RoboDK station: 03 - Palletizing.rdk

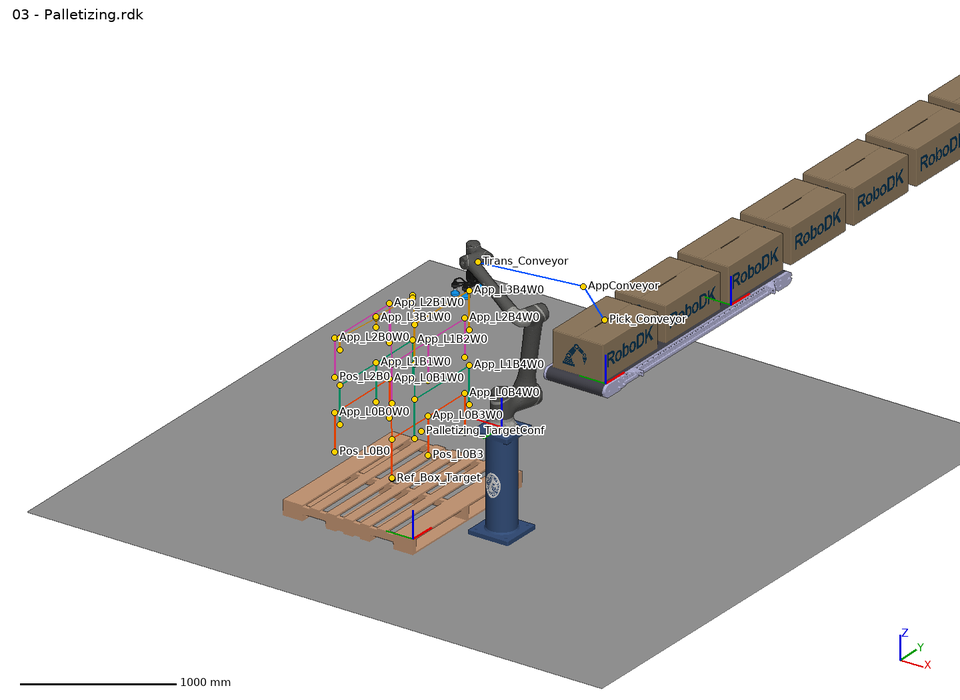
[picture v0: the station drawn from its stored meshes, robots at their saved joint values, targets as dots, program paths as lines]
Station 03 - Palletizing (saved by RoboDK 5.2.4). Poses are relative to the parent item; angles as X-Y-Z fixed-axis rotations.
Station parameters (name, value as stored): Conv_Run, 0, IO_5, 1
  - frame Omron TM12X Base at (0, 0, 0) mm, rotated rx 0 ry 0 rz 180 deg
    - object Pedestal H12in at (0, 0, -305) mm, rotated rx 0 ry 0 rz -90 deg, size 320 x 320 x 304.8 mm, geometry from Pedestal-H12in (2).sld
    - object Pedestal H24in at (0, 0, 0) mm, rotated rx 0 ry 0 rz -180 deg, size 312.1 x 312.1 x 743.1 mm, geometry from Pedestal-H24in.sld
    - object Box 24X16 at (0, 0, 0) mm, size 398.1 x 610.2 x 267.5 mm, geometry from Box 24x16 closed.step
    - robot Omron TM12X: 6 axes, payload 12 kg, reach 1300 mm, repeatability 0.1 mm, weight 33.3 kg
        modified DH rows (alpha deg, a mm, theta deg, d mm): 0, 0, 0, 165.2; 90, 0, 90, 0; 0, 636.1, 0, 0; 0, 557.9, -90, 156.3; -90, 0, 0, 106; 90, 0, 180, 113.15
        joint limits [-125, -90, -60, -145, 0, -200] to [90, 130, 166, 90, 180, 125]; home [0, 0, 90, 0, 90, 0]; saved at [-17.678, -9.72, 76.178, 23.542, 90, -17.678]
      - tool RobotiQ EPick Four, TCP at (0, 30, 180) mm, size 239 x 147 x 184.9 mm
    - frame Conveyor Belt Base at (-430, -550, 210) mm, rotated rx 0 ry 0 rz -90 deg
      - robot Conveyor Belt: 1 axes
          modified DH rows (alpha deg, a mm, theta deg, d mm): 0, 0, 0, 0 linear
          base shift (0, 0, 0) mm, rotated rx 0 ry 90 rz 0 deg
          joint limits [-500000] to [500000]; home [0]; saved at [0]
        - frame Conveyor Box at (0, 0, 0) mm
          - object Box_24X16 at (700, 420, 0) mm, rotated rx 0 ry 0 rz -90 deg, size 398.1 x 610.2 x 267.5 mm, geometry from Box 24x16 closed.step
          - object Box_24X16 at (1400, 420, 0) mm, rotated rx 0 ry 0 rz -90 deg, size 398.1 x 610.2 x 267.5 mm, geometry from Box 24x16 closed.step
          - object Box_24X16 at (5600, 420, 0) mm, rotated rx 0 ry 0 rz -90 deg, size 398.1 x 610.2 x 267.5 mm, geometry from Box 24x16 closed.step
          - object Box_24X16 at (6300, 420, 0) mm, rotated rx 0 ry 0 rz -90 deg, size 398.1 x 610.2 x 267.5 mm, geometry from Box 24x16 closed.step
          - object Box_24X16 at (7700, 420, 0) mm, rotated rx 0 ry 0 rz -90 deg, size 398.1 x 610.2 x 267.5 mm, geometry from Box 24x16 closed.step
          - object Box_24X16 at (7000, 420, 0) mm, rotated rx 0 ry 0 rz -90 deg, size 398.1 x 610.2 x 267.5 mm, geometry from Box 24x16 closed.step
          - object Box_24X16 at (8400, 420, 0) mm, rotated rx 0 ry 0 rz -90 deg, size 398.1 x 610.2 x 267.5 mm, geometry from Box 24x16 closed.step
          - object Box_24X16 at (9100, 420, 0) mm, rotated rx 0 ry 0 rz -90 deg, size 398.1 x 610.2 x 267.5 mm, geometry from Box 24x16 closed.step
          - object Box_24X16 at (10500, 420, 0) mm, rotated rx 0 ry 0 rz -90 deg, size 398.1 x 610.2 x 267.5 mm, geometry from Box 24x16 closed.step
          - object Box_24X16 at (9800, 420, 0) mm, rotated rx 0 ry 0 rz -90 deg, size 398.1 x 610.2 x 267.5 mm, geometry from Box 24x16 closed.step
          - object Box_24X16 at (11200, 420, 0) mm, rotated rx 0 ry 0 rz -90 deg, size 398.1 x 610.2 x 267.5 mm, geometry from Box 24x16 closed.step
          - object Box_24X16 at (11900, 420, 0) mm, rotated rx 0 ry 0 rz -90 deg, size 398.1 x 610.2 x 267.5 mm, geometry from Box 24x16 closed.step
          - object Box_24X16 at (13300, 420, 0) mm, rotated rx 0 ry 0 rz -90 deg, size 398.1 x 610.2 x 267.5 mm, geometry from Box 24x16 closed.step
          - object Box_24X16 at (12600, 420, 0) mm, rotated rx 0 ry 0 rz -90 deg, size 398.1 x 610.2 x 267.5 mm, geometry from Box 24x16 closed.step
          - object Box_24X16 at (0, 420, 0) mm, rotated rx 0 ry 0 rz -90 deg, size 398.1 x 610.2 x 267.5 mm, geometry from Box 24x16 closed.step
          - object Box_24X16 at (2800, 420, 0) mm, rotated rx 0 ry 0 rz -90 deg, size 398.1 x 610.2 x 267.5 mm, geometry from Box 24x16 closed.step
          - object Box_24X16 at (2100, 420, 0) mm, rotated rx 0 ry 0 rz -90 deg, size 398.1 x 610.2 x 267.5 mm, geometry from Box 24x16 closed.step
          - object Box_24X16 at (3500, 420, 0) mm, rotated rx 0 ry 0 rz -90 deg, size 398.1 x 610.2 x 267.5 mm, geometry from Box 24x16 closed.step
          - object Box_24X16 at (4900, 420, 0) mm, rotated rx 0 ry 0 rz -90 deg, size 398.1 x 610.2 x 267.5 mm, geometry from Box 24x16 closed.step
          - object Box_24X16 at (4200, 420, 0) mm, rotated rx 0 ry 0 rz -90 deg, size 398.1 x 610.2 x 267.5 mm, geometry from Box 24x16 closed.step
      - target AppConveyor (Cartesian target) at (69.16, 222.69, 602.66) mm, rotated rx 180 ry 0 rz 179.98 deg; joints [-97.337, 6.658, 49.734, 33.608, 90, -97.317, 0] of Omron TM12X
      - target Pick_Conveyor (Cartesian target) at (304.16, 222.6, 268.74) mm, rotated rx 180 ry 0 rz 179.98 deg; joints [-95.378, 19.16, 70.241, 0.599, 90, -95.357, 0] of Omron TM12X
      - target Trans_Conveyor (Cartesian target) at (-198.64, 863.17, 703.7) mm, rotated rx 180 ry 0 rz -107.24 deg; joints [-25.922, 5.576, 37.342, 47.082, 90, -98.682] of Omron TM12X
      - frame New_Box 24X16 at (1400, 0, 0) mm
        - object BoxRef_24X16 at (0, 420, 0) mm, rotated rx 0 ry 0 rz -90 deg, size 398.1 x 610.2 x 267.5 mm, geometry from Box 24x16 closed.step
    - frame Pallet at (268.35, 609.6, -630.58) mm, rotated rx 0 ry 0 rz -90 deg
      - object Pallet 40inx48in at (0, 0, 0) mm, size 1219.2 x 1016 x 114.3 mm, geometry from AR3.step
      - target Ref_Box_Target (Cartesian target) at (198.15, 304.17, 268.74) mm, rotated rx -180 ry 0 rz -90 deg; joints [46.804, 34.313, 124.082, -68.396, 90, -43.196] of Omron TM12X
      - target Palletizing_TargetConfig (Cartesian target) at (676.2, 408.21, 385.47) mm, rotated rx -179.16 ry 1.93 rz -48.82 deg; joints [5.592, 37.489, 126.42, -75.963, 90.438, -125.563] of Omron TM12X
      - folder Palletizing_Data: PalletData
        - folder Palletizing_Data_L0: PalletData
          - target App_L0B0W0 (Cartesian target) at (303.25, 822.47, 550) mm, rotated rx -180 ry 0 rz -180 deg; joints [24.246, 55.576, 68.456, -34.032, 90, 24.246] of Omron TM12X
          - target Ret_L0B0W0 (Cartesian target) at (303.25, 822.47, 550) mm, rotated rx -180 ry 0 rz -180 deg; joints [24.246, 55.576, 68.456, -34.032, 90, 24.246] of Omron TM12X
          - target Pos_L0B0 (Cartesian target) at (303.25, 822.47, 270) mm, rotated rx -180 ry 0 rz -180 deg; joints [24.246, 73.661, 63.877, -47.538, 90, 24.246] of Omron TM12X
          - target App_L0B1W0 (Cartesian target) at (913.41, 822.47, 550) mm, rotated rx -180 ry 0 rz -180 deg; joints [-7.838, 55.519, 68.577, -34.096, 90, -7.838] of Omron TM12X
          - target Ret_L0B1W0 (Cartesian target) at (913.41, 822.47, 550) mm, rotated rx -180 ry 0 rz -180 deg; joints [-7.838, 55.519, 68.577, -34.096, 90, -7.838] of Omron TM12X
          - target Pos_L0B1 (Cartesian target) at (913.41, 822.47, 270) mm, rotated rx -180 ry 0 rz -180 deg; joints [-7.838, 73.613, 64.003, -47.616, 90, -7.838] of Omron TM12X
          - target App_L0B2W0 (Cartesian target) at (197.9, 303.25, 550) mm, rotated rx -180 ry 0 rz -90 deg; joints [46.878, 30.236, 123.942, -64.178, 90, -43.122] of Omron TM12X
          - target Ret_L0B2W0 (Cartesian target) at (197.9, 303.25, 550) mm, rotated rx -180 ry 0 rz -90 deg; joints [46.878, 30.236, 123.942, -64.178, 90, -43.122] of Omron TM12X
          - target Pos_L0B2 (Cartesian target) at (197.9, 303.25, 270) mm, rotated rx -180 ry 0 rz -90 deg; joints [46.878, 59.272, 119.029, -88.302, 90, -43.122] of Omron TM12X
          - target App_L0B3W0 (Cartesian target) at (604.3, 303.25, 550) mm, rotated rx -180 ry 0 rz -90 deg; joints [13.38, 24.947, 136.655, -71.602, 90, -76.62] of Omron TM12X
          - target Ret_L0B3W0 (Cartesian target) at (604.3, 303.25, 550) mm, rotated rx -180 ry 0 rz -90 deg; joints [13.38, 24.947, 136.655, -71.602, 90, -76.62] of Omron TM12X
          - target Pos_L0B3 (Cartesian target) at (604.3, 303.25, 270) mm, rotated rx -180 ry 0 rz -90 deg; joints [13.38, 60.356, 130.855, -101.211, 90, -76.62] of Omron TM12X
          - target App_L0B4W0 (Cartesian target) at (1015.06, 303.25, 550) mm, rotated rx -180 ry 0 rz -90 deg; joints [-24.738, 31.775, 120.399, -62.175, 90, -114.738] of Omron TM12X
          - target Ret_L0B4W0 (Cartesian target) at (1015.06, 303.25, 550) mm, rotated rx -180 ry 0 rz -90 deg; joints [-24.738, 31.775, 120.399, -62.175, 90, -114.738] of Omron TM12X
          - target Pos_L0B4 (Cartesian target) at (1015.06, 303.25, 270) mm, rotated rx -180 ry 0 rz -90 deg; joints [-24.738, 59.459, 115.654, -85.113, 90, -114.738] of Omron TM12X
        - folder Palletizing_Data_L1: PalletData
          - target App_L1B0W0 (Cartesian target) at (197.9, 709.65, 817.48) mm, rotated rx -180 ry 0 rz -90 deg; joints [29.882, 39.329, 69.189, -18.518, 90, -60.118] of Omron TM12X
          - target Ret_L1B0W0 (Cartesian target) at (197.9, 709.65, 817.48) mm, rotated rx -180 ry 0 rz -90 deg; joints [29.882, 39.329, 69.189, -18.518, 90, -60.118] of Omron TM12X
          - target Pos_L1B0 (Cartesian target) at (197.9, 709.65, 537.48) mm, rotated rx -180 ry 0 rz -90 deg; joints [29.882, 52.141, 77.448, -39.589, 90, -60.118] of Omron TM12X
          - target App_L1B1W0 (Cartesian target) at (604.3, 709.65, 817.48) mm, rotated rx -180 ry 0 rz -90 deg; joints [7.747, 33.003, 80.067, -23.07, 90, -82.253] of Omron TM12X
          - target Ret_L1B1W0 (Cartesian target) at (604.3, 709.65, 817.48) mm, rotated rx -180 ry 0 rz -90 deg; joints [7.747, 33.003, 80.067, -23.07, 90, -82.253] of Omron TM12X
          - target Pos_L1B1 (Cartesian target) at (604.3, 709.65, 537.48) mm, rotated rx -180 ry 0 rz -90 deg; joints [7.747, 47.289, 88.021, -45.31, 90, -82.253] of Omron TM12X
          - target App_L1B2W0 (Cartesian target) at (1015.06, 709.65, 817.48) mm, rotated rx -180 ry 0 rz -90 deg; joints [-15.606, 41.274, 65.737, -17.012, 90, -105.606] of Omron TM12X
          - target Ret_L1B2W0 (Cartesian target) at (1015.06, 709.65, 817.48) mm, rotated rx -180 ry 0 rz -90 deg; joints [-15.606, 41.274, 65.737, -17.012, 90, -105.606] of Omron TM12X
          - target Pos_L1B2 (Cartesian target) at (1015.06, 709.65, 537.48) mm, rotated rx -180 ry 0 rz -90 deg; joints [-15.606, 53.66, 74.159, -37.819, 90, -105.606] of Omron TM12X
          - target App_L1B3W0 (Cartesian target) at (303.25, 200.17, 817.48) mm, rotated rx -180 ry 0 rz -180 deg; joints [51.927, -4.692, 129.582, -34.89, 90, 51.927] of Omron TM12X
          - target Ret_L1B3W0 (Cartesian target) at (303.25, 200.17, 817.48) mm, rotated rx -180 ry 0 rz -180 deg; joints [51.927, -4.692, 129.582, -34.89, 90, 51.927] of Omron TM12X
          - target Pos_L1B3 (Cartesian target) at (303.25, 200.17, 537.48) mm, rotated rx -180 ry 0 rz -180 deg; joints [51.927, 25.107, 140.818, -75.925, 90, 51.927] of Omron TM12X
          - target App_L1B4W0 (Cartesian target) at (913.41, 200.17, 817.48) mm, rotated rx -180 ry 0 rz -180 deg; joints [-17.678, -4.838, 129.711, -34.873, 90, -17.678] of Omron TM12X
          - target Ret_L1B4W0 (Cartesian target) at (913.41, 200.17, 817.48) mm, rotated rx -180 ry 0 rz -180 deg; joints [-17.678, -4.838, 129.711, -34.873, 90, -17.678] of Omron TM12X
          - target Pos_L1B4 (Cartesian target) at (913.41, 200.17, 537.48) mm, rotated rx -180 ry 0 rz -180 deg; joints [-17.678, 25.055, 140.975, -76.03, 90, -17.678] of Omron TM12X
        - folder Palletizing_Data_L2: PalletData
          - target App_L2B0W0 (Cartesian target) at (303.25, 822.47, 1084.96) mm, rotated rx -180 ry 0 rz -180 deg; joints [24.246, 44.227, 32.666, 13.106, 90, 24.246] of Omron TM12X
          - target Ret_L2B0W0 (Cartesian target) at (303.25, 822.47, 1084.96) mm, rotated rx -180 ry 0 rz -180 deg; joints [24.246, 44.227, 32.666, 13.106, 90, 24.246] of Omron TM12X
          - target Pos_L2B0 (Cartesian target) at (303.25, 822.47, 804.96) mm, rotated rx -180 ry 0 rz -180 deg; joints [24.246, 44.92, 60.473, -15.393, 90, 24.246] of Omron TM12X
          - target App_L2B1W0 (Cartesian target) at (913.41, 822.47, 1084.96) mm, rotated rx -180 ry 0 rz -180 deg; joints [-7.838, 44.112, 32.875, 13.013, 90, -7.838] of Omron TM12X
          - target Ret_L2B1W0 (Cartesian target) at (913.41, 822.47, 1084.96) mm, rotated rx -180 ry 0 rz -180 deg; joints [-7.838, 44.112, 32.875, 13.013, 90, -7.838] of Omron TM12X
          - target Pos_L2B1 (Cartesian target) at (913.41, 822.47, 804.96) mm, rotated rx -180 ry 0 rz -180 deg; joints [-7.838, 44.849, 60.603, -15.452, 90, -7.838] of Omron TM12X
          - target App_L2B2W0 (Cartesian target) at (197.9, 303.25, 1084.96) mm, rotated rx -180 ry 0 rz -90 deg; joints [46.878, 0.723, 94.803, -5.526, 90, -43.122] of Omron TM12X
          - target Ret_L2B2W0 (Cartesian target) at (197.9, 303.25, 1084.96) mm, rotated rx -180 ry 0 rz -90 deg; joints [46.878, 0.723, 94.803, -5.526, 90, -43.122] of Omron TM12X
          - target Pos_L2B2 (Cartesian target) at (197.9, 303.25, 804.96) mm, rotated rx -180 ry 0 rz -90 deg; joints [46.878, 9.9, 115.641, -35.541, 90, -43.122] of Omron TM12X
          - target App_L2B3W0 (Cartesian target) at (604.3, 303.25, 1084.96) mm, rotated rx -180 ry 0 rz -90 deg; joints [13.38, -10.122, 104.633, -4.51, 90, -76.62] of Omron TM12X
          - target Ret_L2B3W0 (Cartesian target) at (604.3, 303.25, 1084.96) mm, rotated rx -180 ry 0 rz -90 deg; joints [13.38, -10.122, 104.633, -4.51, 90, -76.62] of Omron TM12X
          - target Pos_L2B3 (Cartesian target) at (604.3, 303.25, 804.96) mm, rotated rx -180 ry 0 rz -90 deg; joints [13.38, -0.241, 126.986, -36.745, 90, -76.62] of Omron TM12X
          - target App_L2B4W0 (Cartesian target) at (1015.06, 303.25, 1084.96) mm, rotated rx -180 ry 0 rz -90 deg; joints [-24.738, 3.601, 91.8, -5.401, 90, -114.738] of Omron TM12X
          - target Ret_L2B4W0 (Cartesian target) at (1015.06, 303.25, 1084.96) mm, rotated rx -180 ry 0 rz -90 deg; joints [-24.738, 3.601, 91.8, -5.401, 90, -114.738] of Omron TM12X
          - target Pos_L2B4 (Cartesian target) at (1015.06, 303.25, 804.96) mm, rotated rx -180 ry 0 rz -90 deg; joints [-24.738, 12.483, 112.359, -34.842, 90, -114.738] of Omron TM12X
        - folder Palletizing_Data_L3: PalletData
          - target App_L3B0W0 (Cartesian target) at (197.9, 709.65, 1150.44) mm, rotated rx -180 ry 0 rz -90 deg; joints [29.882, 38.325, 36.209, 15.467, 90, -60.118] of Omron TM12X
          - target Ret_L3B0W0 (Cartesian target) at (197.9, 709.65, 1158.34) mm, rotated rx -180 ry 0 rz -90 deg; joints [29.882, 38.663, 34.775, 16.561, 90, -60.118] of Omron TM12X
          - target Pos_L3B0 (Cartesian target) at (197.9, 709.65, 1072.44) mm, rotated rx -180 ry 0 rz -90 deg; joints [29.882, 36.374, 47.696, 5.93, 90, -60.118] of Omron TM12X
          - target App_L3B1W0 (Cartesian target) at (604.3, 709.65, 1137.62) mm, rotated rx -180 ry 0 rz -90 deg; joints [7.747, 28.892, 53.064, 8.044, 90, -82.253] of Omron TM12X
          - target Ret_L3B1W0 (Cartesian target) at (604.3, 709.65, 1148.74) mm, rotated rx -180 ry 0 rz -90 deg; joints [7.747, 29.083, 51.611, 9.306, 90, -82.253] of Omron TM12X
          - target Pos_L3B1 (Cartesian target) at (604.3, 709.65, 1072.44) mm, rotated rx -180 ry 0 rz -90 deg; joints [7.747, 28.338, 60.641, 1.021, 90, -82.253] of Omron TM12X
          - target App_L3B2W0 (Cartesian target) at (1015.06, 709.65, 1132.36) mm, rotated rx -180 ry 0 rz -90 deg; joints [-15.606, 40.738, 33.904, 15.357, 90, -105.606] of Omron TM12X
          - target Ret_L3B2W0 (Cartesian target) at (1015.06, 709.65, 1116.88) mm, rotated rx -180 ry 0 rz -90 deg; joints [-15.606, 40.141, 36.599, 13.26, 90, -105.606] of Omron TM12X
          - target Pos_L3B2 (Cartesian target) at (1015.06, 709.65, 1072.44) mm, rotated rx -180 ry 0 rz -90 deg; joints [-15.606, 39.002, 43.222, 7.776, 90, -105.606] of Omron TM12X
          - target App_L3B3W0 (Cartesian target) at (303.25, 200.17, 1352.44) mm, rotated rx -180 ry 0 rz -180 deg; joints [51.927, -9.591, 76.076, 23.515, 90, 51.927] of Omron TM12X
          - target Ret_L3B3W0 (Cartesian target) at (303.25, 200.17, 1352.44) mm, rotated rx -180 ry 0 rz -180 deg; joints [51.927, -9.591, 76.076, 23.515, 90, 51.927] of Omron TM12X
          - target Pos_L3B3 (Cartesian target) at (303.25, 200.17, 1072.44) mm, rotated rx -180 ry 0 rz -180 deg; joints [51.927, -13.66, 108.627, -4.967, 90, 51.927] of Omron TM12X
          - target App_L3B4W0 (Cartesian target) at (913.41, 200.17, 1352.44) mm, rotated rx -180 ry 0 rz -180 deg; joints [-17.678, -9.72, 76.178, 23.542, 90, -17.678] of Omron TM12X
          - target Ret_L3B4W0 (Cartesian target) at (913.41, 200.17, 1352.44) mm, rotated rx -180 ry 0 rz -180 deg; joints [-17.678, -9.72, 76.178, 23.542, 90, -17.678] of Omron TM12X
          - target Pos_L3B4 (Cartesian target) at (913.41, 200.17, 1072.44) mm, rotated rx -180 ry 0 rz -180 deg; joints [-17.678, -13.804, 108.731, -4.928, 90, -17.678] of Omron TM12X
    - object Floor at (410, -740, -746) mm, rotated rx 0 ry 0 rz -180 deg, size 4500 x 4500 x 0 mm, geometry from Floor.sld
  - program Pick_Box (16 instructions, listed below)
  - program Drop_Box (1 instructions, listed below)
  - program Conv_Move_Sync (3 instructions, listed below)
  - program Init (3 instructions, listed below)
  - folder Python
    - Python program Clear_Conveyor (listed below)
    - Python program Clear_Pallet (listed below)
    - Python program Clear_Tool (listed below)
    - Python program Conv_Init_Position (listed below)
    - Python program Conv_Move_24X16 (listed below)
    - Python program New_Box_24X16 (listed below)
  - item type 20 Palletizing Settings: svg | Palletizing Plugin | Pallet | Box | Box | Box | Box | Init | Pick_Box | Drop_Box | Layer_%1 | OnFinish | Palletizing_TargetConfig | Palletizing | Pos_L%1_B%2 | App_L%1_B%2 | RunTask | Layer_%LAYER_NUM%_End | Ret_L%1_B%2_W%3
  - program Replace_Objects (1 instructions, listed below)
  - folder Palletizing_Progs: PalletData
    - program Palletizing_Main (5 instructions, listed below)
    - program Palletizing_L0 (60 instructions, listed below)
    - program Palletizing_L1 (60 instructions, listed below)
    - program Palletizing_L2 (60 instructions, listed below)
    - program Palletizing_L3 (60 instructions, listed below)
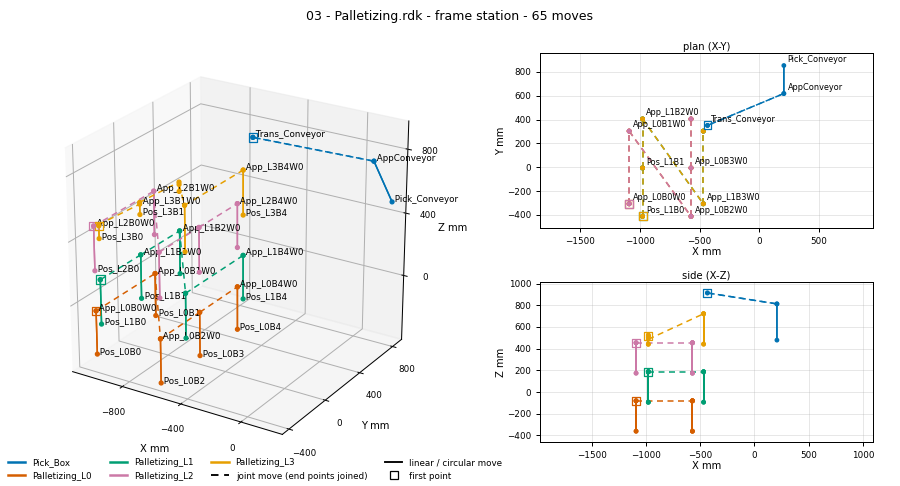
[picture p0: tool path of 03 - Palletizing.rdk in frame station, 65 of 65 moves have a stored position in this frame; points joined in program order, loops and branches not executed]

--- program Pick_Box (robot Omron TM12X) ---
  Set Ref.: Conveyor Belt Base
  Set Tool: RobotiQ EPick Four
  Set speed (500.0 mm/s)
  Smooth(10)
  MoveJ (Trans_Conveyor)
  MoveJ (AppConveyor)
  Wait Conv_Run=0
  Set speed (200.0 mm/s)
  Accurate (rounding -1 mm)
  MoveL (Pick_Conveyor)
  Attach to RobotiQ EPick Four
  Set speed (500.0 mm/s)
  Smooth(10)
  MoveL (AppConveyor)
  Run Conv_Move_Sync
  MoveJ (Trans_Conveyor)

--- program Drop_Box (robot Omron TM12X) ---
  Detach from RobotiQ EPick Four

--- program Conv_Move_Sync (robot Omron TM12X) ---
  Set Conv_Run=1
  Call Conv_Move_24X16
  Set Conv_Run=0

--- program Init (robot Omron TM12X) ---
  Call Conv_Init_Position
  Call Replace_Objects
  Set Conv_Run=0

--- Python program Clear_Conveyor ---
# Type help("robolink") or help("robodk") for more information
# Press F5 to run the script
# Documentation: https://robodk.com/doc/en/RoboDK-API.html
# Reference:     https://robodk.com/doc/en/PythonAPI/index.html
# Note: It is not required to keep a copy of this file, your python script is saved with the station
from robolink import *    # RoboDK API
from robodk import *      # Robot toolbox
RDK = Robolink()

#----- CONSTANT -----
CONV_FRAME_NAME = 'Conveyor Box'

#----- PROGRAM -----
frame = RDK.Item(CONV_FRAME_NAME,ITEM_TYPE_FRAME)

if frame.Valid():
    for item in frame.Childs():
        if item.Type() == ITEM_TYPE_OBJECT:
            item.Delete()

--- Python program Clear_Pallet ---
# Type help("robolink") or help("robodk") for more information
# Press F5 to run the script
# Documentation: https://robodk.com/doc/en/RoboDK-API.html
# Reference:     https://robodk.com/doc/en/PythonAPI/index.html
# Note: It is not required to keep a copy of this file, your python script is saved with the station
from robolink import *    # RoboDK API
from robodk import *      # Robot toolbox
RDK = Robolink()

#----- CONSTANT -----
FRAME_NAME = 'Pallet'

#----- PROGRAM -----
frame = RDK.Item(FRAME_NAME,ITEM_TYPE_FRAME)

if frame.Valid():
    for item in frame.Childs():
        if item.Type() == ITEM_TYPE_OBJECT:
            if not item.Name().lower().startswith('pallet'):
                item.Delete()

--- Python program Clear_Tool ---
# Type help("robolink") or help("robodk") for more information
# Press F5 to run the script
# Documentation: https://robodk.com/doc/en/RoboDK-API.html
# Reference:     https://robodk.com/doc/en/PythonAPI/index.html
# Note: It is not required to keep a copy of this file, your python script is saved with the station
from robolink import *    # RoboDK API
from robodk import *      # Robot toolbox
RDK = Robolink()

#----- CONSTANT -----
TOOL_NAME = 'RobotiQ EPick Four'

#----- PROGRAM -----
tool = RDK.Item(TOOL_NAME,ITEM_TYPE_TOOL)

if tool.Valid():
    for item in tool.Childs():
        if item.Type() == ITEM_TYPE_OBJECT:
            item.Delete()

--- Python program Conv_Init_Position ---
# Type help("robolink") or help("robodk") for more information
# Press F5 to run the script
# Documentation: https://robodk.com/doc/en/RoboDK-API.html
# Reference:     https://robodk.com/doc/en/PythonAPI/index.html
# Note: It is not required to keep a copy of this file, your python script is saved with the station
from robolink import *    # RoboDK API
from robodk import *      # Robot toolbox
RDK = Robolink()

MECHANISM_NAME = 'Conveyor Belt'
mechanism = RDK.Item(MECHANISM_NAME,itemtype=ITEM_TYPE_ROBOT)

if mechanism.Valid():
    mechanism.setJoints([0])

--- Python program Conv_Move_24X16 ---
# Type help("robolink") or help("robodk") for more information
# Press F5 to run the script
# Documentation: https://robodk.com/doc/en/RoboDK-API.html
# Reference:     https://robodk.com/doc/en/PythonAPI/index.html
# Note: It is not required to keep a copy of this file, your python script is saved with the station
from robolink import *    # RoboDK API
from robodk import *      # Robot toolbox
RDK = Robolink()

#------ CONSTANT ------
MECHANISM_NAME = 'Conveyor Belt'
PART_TRAVEL_MM = -700

mechanism = RDK.Item(MECHANISM_NAME,itemtype=ITEM_TYPE_ROBOT)

if mechanism.Valid():
    mechanism.MoveJ(mechanism.Joints() + PART_TRAVEL_MM)

--- Python program New_Box_24X16 ---
# Type help("robolink") or help("robodk") for more information
# Press F5 to run the script
# Documentation: https://robodk.com/doc/en/RoboDK-API.html
# Reference:     https://robodk.com/doc/en/PythonAPI/index.html
# Note: It is not required to keep a copy of this file, your python script is saved with the station
from robolink import *    # RoboDK API
from robodk import *      # Robot toolbox
RDK = Robolink()



#----- Constante -----
NEW_REF_OBJECT_NAME = 'BoxRef_24X16'
NEW_OBJECT_NAME = 'Box_24X16'
REFERENCE_FRAME = 'Conveyor Box'
REFERENCE_FRAME_REF = 'New_Box 24X16'


#------- Program ------
frame = RDK.Item(REFERENCE_FRAME, ITEM_TYPE_FRAME)
frame_ref = RDK.Item(REFERENCE_FRAME_REF, ITEM_TYPE_FRAME)
ref_obj = RDK.Item(NEW_REF_OBJECT_NAME, ITEM_TYPE_OBJECT)

RDK.Render(False)
if frame.Valid() and  ref_obj.Valid():
    ref_obj.Copy()
    new_obj = RDK.Paste()
    new_obj.setVisible(False)
    new_obj.setName(NEW_OBJECT_NAME)
    new_obj.setParent(frame_ref)
    RDK.Update()
    new_obj.setParentStatic(frame)
    new_obj.setVisible(True)
RDK.Render(True)

--- program Replace_Objects (robot Omron TM12X) ---
  Replace objects

--- program Palletizing_Main (robot Omron TM12X) ---
  Call Init
  Call Palletizing_L0
  Call Palletizing_L1
  Call Palletizing_L2
  Call Palletizing_L3

--- program Palletizing_L0 (robot Omron TM12X) ---
  Call Pick_Box
  Set Ref.: Pallet
  Smooth(10)
  Set speed (100.0 mm/s)
  MoveJ (App_L0B0W0)
  Accurate (rounding -1 mm)
  MoveL (Pos_L0B0)
  Call Drop_Box
  Set Ref.: Pallet
  Smooth(10)
  Set speed (250.0 mm/s)
  MoveL (Ret_L0B0W0)
  Call Pick_Box
  Set Ref.: Pallet
  Smooth(10)
  Set speed (100.0 mm/s)
  MoveJ (App_L0B1W0)
  Accurate (rounding -1 mm)
  MoveL (Pos_L0B1)
  Call Drop_Box
  Set Ref.: Pallet
  Smooth(10)
  Set speed (250.0 mm/s)
  MoveL (Ret_L0B1W0)
  Call Pick_Box
  Set Ref.: Pallet
  Smooth(10)
  Set speed (100.0 mm/s)
  MoveJ (App_L0B2W0)
  Accurate (rounding -1 mm)
  MoveL (Pos_L0B2)
  Call Drop_Box
  Set Ref.: Pallet
  Smooth(10)
  Set speed (250.0 mm/s)
  MoveL (Ret_L0B2W0)
  Call Pick_Box
  Set Ref.: Pallet
  Smooth(10)
  Set speed (100.0 mm/s)
  MoveJ (App_L0B3W0)
  Accurate (rounding -1 mm)
  MoveL (Pos_L0B3)
  Call Drop_Box
  Set Ref.: Pallet
  Smooth(10)
  Set speed (250.0 mm/s)
  MoveL (Ret_L0B3W0)
  Call Pick_Box
  Set Ref.: Pallet
  Smooth(10)
  Set speed (100.0 mm/s)
  MoveJ (App_L0B4W0)
  Accurate (rounding -1 mm)
  MoveL (Pos_L0B4)
  Call Drop_Box
  Set Ref.: Pallet
  Smooth(10)
  Set speed (250.0 mm/s)
  MoveL (Ret_L0B4W0)

--- program Palletizing_L1 (robot Omron TM12X) ---
  Call Pick_Box
  Set Ref.: Pallet
  Smooth(10)
  Set speed (100.0 mm/s)
  MoveJ (App_L1B0W0)
  Accurate (rounding -1 mm)
  MoveL (Pos_L1B0)
  Call Drop_Box
  Set Ref.: Pallet
  Smooth(10)
  Set speed (250.0 mm/s)
  MoveL (Ret_L1B0W0)
  Call Pick_Box
  Set Ref.: Pallet
  Smooth(10)
  Set speed (100.0 mm/s)
  MoveJ (App_L1B1W0)
  Accurate (rounding -1 mm)
  MoveL (Pos_L1B1)
  Call Drop_Box
  Set Ref.: Pallet
  Smooth(10)
  Set speed (250.0 mm/s)
  MoveL (Ret_L1B1W0)
  Call Pick_Box
  Set Ref.: Pallet
  Smooth(10)
  Set speed (100.0 mm/s)
  MoveJ (App_L1B2W0)
  Accurate (rounding -1 mm)
  MoveL (Pos_L1B2)
  Call Drop_Box
  Set Ref.: Pallet
  Smooth(10)
  Set speed (250.0 mm/s)
  MoveL (Ret_L1B2W0)
  Call Pick_Box
  Set Ref.: Pallet
  Smooth(10)
  Set speed (100.0 mm/s)
  MoveJ (App_L1B3W0)
  Accurate (rounding -1 mm)
  MoveL (Pos_L1B3)
  Call Drop_Box
  Set Ref.: Pallet
  Smooth(10)
  Set speed (250.0 mm/s)
  MoveL (Ret_L1B3W0)
  Call Pick_Box
  Set Ref.: Pallet
  Smooth(10)
  Set speed (100.0 mm/s)
  MoveJ (App_L1B4W0)
  Accurate (rounding -1 mm)
  MoveL (Pos_L1B4)
  Call Drop_Box
  Set Ref.: Pallet
  Smooth(10)
  Set speed (250.0 mm/s)
  MoveL (Ret_L1B4W0)

--- program Palletizing_L2 (robot Omron TM12X) ---
  Call Pick_Box
  Set Ref.: Pallet
  Smooth(10)
  Set speed (100.0 mm/s)
  MoveJ (App_L2B0W0)
  Accurate (rounding -1 mm)
  MoveL (Pos_L2B0)
  Call Drop_Box
  Set Ref.: Pallet
  Smooth(10)
  Set speed (250.0 mm/s)
  MoveL (Ret_L2B0W0)
  Call Pick_Box
  Set Ref.: Pallet
  Smooth(10)
  Set speed (100.0 mm/s)
  MoveJ (App_L2B1W0)
  Accurate (rounding -1 mm)
  MoveL (Pos_L2B1)
  Call Drop_Box
  Set Ref.: Pallet
  Smooth(10)
  Set speed (250.0 mm/s)
  MoveL (Ret_L2B1W0)
  Call Pick_Box
  Set Ref.: Pallet
  Smooth(10)
  Set speed (100.0 mm/s)
  MoveJ (App_L2B2W0)
  Accurate (rounding -1 mm)
  MoveL (Pos_L2B2)
  Call Drop_Box
  Set Ref.: Pallet
  Smooth(10)
  Set speed (250.0 mm/s)
  MoveL (Ret_L2B2W0)
  Call Pick_Box
  Set Ref.: Pallet
  Smooth(10)
  Set speed (100.0 mm/s)
  MoveJ (App_L2B3W0)
  Accurate (rounding -1 mm)
  MoveL (Pos_L2B3)
  Call Drop_Box
  Set Ref.: Pallet
  Smooth(10)
  Set speed (250.0 mm/s)
  MoveL (Ret_L2B3W0)
  Call Pick_Box
  Set Ref.: Pallet
  Smooth(10)
  Set speed (100.0 mm/s)
  MoveJ (App_L2B4W0)
  Accurate (rounding -1 mm)
  MoveL (Pos_L2B4)
  Call Drop_Box
  Set Ref.: Pallet
  Smooth(10)
  Set speed (250.0 mm/s)
  MoveL (Ret_L2B4W0)

--- program Palletizing_L3 (robot Omron TM12X) ---
  Call Pick_Box
  Set Ref.: Pallet
  Smooth(10)
  Set speed (100.0 mm/s)
  MoveJ (App_L3B0W0)
  Accurate (rounding -1 mm)
  MoveL (Pos_L3B0)
  Call Drop_Box
  Set Ref.: Pallet
  Smooth(10)
  Set speed (250.0 mm/s)
  MoveL (Ret_L3B0W0)
  Call Pick_Box
  Set Ref.: Pallet
  Smooth(10)
  Set speed (100.0 mm/s)
  MoveJ (App_L3B1W0)
  Accurate (rounding -1 mm)
  MoveL (Pos_L3B1)
  Call Drop_Box
  Set Ref.: Pallet
  Smooth(10)
  Set speed (250.0 mm/s)
  MoveL (Ret_L3B1W0)
  Call Pick_Box
  Set Ref.: Pallet
  Smooth(10)
  Set speed (100.0 mm/s)
  MoveJ (App_L3B2W0)
  Accurate (rounding -1 mm)
  MoveL (Pos_L3B2)
  Call Drop_Box
  Set Ref.: Pallet
  Smooth(10)
  Set speed (250.0 mm/s)
  MoveL (Ret_L3B2W0)
  Call Pick_Box
  Set Ref.: Pallet
  Smooth(10)
  Set speed (100.0 mm/s)
  MoveJ (App_L3B3W0)
  Accurate (rounding -1 mm)
  MoveL (Pos_L3B3)
  Call Drop_Box
  Set Ref.: Pallet
  Smooth(10)
  Set speed (250.0 mm/s)
  MoveL (Ret_L3B3W0)
  Call Pick_Box
  Set Ref.: Pallet
  Smooth(10)
  Set speed (100.0 mm/s)
  MoveJ (App_L3B4W0)
  Accurate (rounding -1 mm)
  MoveL (Pos_L3B4)
  Call Drop_Box
  Set Ref.: Pallet
  Smooth(10)
  Set speed (250.0 mm/s)
  MoveL (Ret_L3B4W0)
